// LS Electric XG5000 project: test1
// PLC NewPLC

PROGRAM NewProgram (task: 스캔 프로그램)

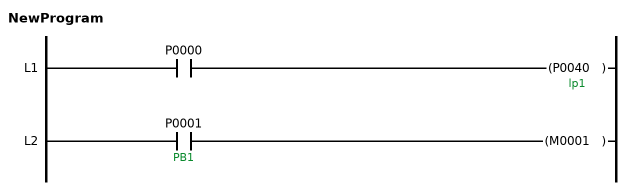
; L1
LOAD      P0000
OUT       P0040	// lp1
; L2
LOAD      P0001	// PB1
OUT       M0001

VARIABLES AND COMMENTS (devices not used above)
P00041	BIT	lp2
P00002	BIT	pb2